FUNCTION_BLOCK SSC_TransferWorkpieceTo_PSStart EXTENDS SSC_MoveWorkpiece_Base
VAR_INPUT
	i_ptrPAC : POINTER TO PicAlphaConveyor;
	i_ptrSSC : POINTER TO SmallSortingConveyor;
END_VAR
VAR_OUTPUT
END_VAR
VAR
	m_ptrPAC : POINTER TO PicAlphaConveyor;
	// (EProcessVariables.PicAlpha_HoldingWorkpiece = FALSE) AND ((EProcessVariables.PicAlpha_CylinderRetracted = TRUE) AND (EProcessVariables.PicAlpha_AtPos4 = TRUE))
	m_compExpr226: ComparisonExpression(EProcessVariables.PicAlpha_HoldingWorkpiece, EComparisonType.equals, EDataType.binary, FALSE, 0, '', TRUE);
	m_compExpr228: ComparisonExpression(EProcessVariables.PicAlpha_CylinderRetracted, EComparisonType.equals, EDataType.binary, TRUE, 0, '', TRUE);
	//m_compExpr230: ComparisonExpression(EProcessVariables.PicAlpha_AtPos4, EComparisonType.equals, EDataType.binary, TRUE, 0, '', TRUE);
	//m_boolExpr231: BoolExpression(m_compExpr228, EBoolOperation.and_op, m_compExpr230);
	m_precondition: BoolExpression(m_compExpr226, EBoolOperation.and_op, m_compExpr228);
	
	// EProcessVariables.SSC_WPAtStart = TRUE
	m_postcondition: ComparisonExpression(EProcessVariables.SSC_WPAtStart, EComparisonType.equals, EDataType.binary, TRUE, 0, '', TRUE);
	m_passby: BOOL;
END_VAR

SUPER^();

METHOD PROTECTED  AtTarget : BOOL
VAR_INPUT
END_VAR
AtTarget := FALSE;

IF m_ptrSSC^.WPAtStart THEN
	m_passby := TRUE;
END_IF

IF m_ptrSSC^.WPAtStart THEN
	m_passby := FALSE;
	AtTarget := TRUE;
END_IF
END_METHOD

METHOD PROTECTED EjectOperation : BOOL
VAR_INPUT
END_VAR
EjectOperation := TRUE;
END_METHOD

METHOD FB_init : BOOL
VAR_INPUT
	bInitRetains : BOOL; // if TRUE, the retain variables are initialized (warm start / cold start)
	bInCopyCode : BOOL;  // if TRUE, the instance afterwards gets moved into the copy code (online change)
	
	i_ptrSSC: POINTER TO SmallSortingConveyor;
	
END_VAR
m_ptrSSC := i_ptrSSC;
m_ptrPAC := i_ptrPAC;
m_passby := FALSE;

m_id := EPrimitives.SSC_TransferWorkpieceTo_PSStart;
m_timeout := T#200S;

Precondition := m_precondition;
Postcondition := m_postcondition;

FB_init := TRUE;
END_METHOD

END_FUNCTION_BLOCK

(* stored: Version 1.1.0.1
   POU SSC_TransferWorkpieceTo_PSStart: Id {828f8b64-2591-43b2-8c9f-9de33114a030}, SpecialFunc None
   Method AtTarget: Id {7a6dfcb4-b6ff-497e-83d7-91e875b5f6b4}
   Method EjectOperation: Id {01af7f4a-74db-4d40-84ac-49a7cd313de8}
   Method FB_init: Id {fc25a999-881b-4674-b79d-05405bd4db72} *)
